{attribute 'GeneratedUsingTerminal: EK1122-0000-0018'}
{attribute addProperty BoxType "EK1122-0000-0018"}
{attribute addProperty Id "Term_17_EK1100Term_17_EK1100_E82441DC140"}
{attribute addProperty CRC "1353770864"}
{attribute addProperty Size "140"}
TYPE Term_16_EK1122_50B0E770 EXTENDS EK1122_1FC0878B :
STRUCT
	{attribute addProperty Name "Term_17_EK1100"}
	{attribute addProperty PreviousPort "Term 16 (EK1122) : D"}
	Term_17_EK1100 : Term_17_EK1100_E82441DC;
END_STRUCT
END_TYPE

(* stored: Version 1.2.0.0, ProductVersion 3.1.4024.9
   DUT Term_16_EK1122_50B0E770: Id {fa7c8029-8d97-0aa7-0914-3c2c5f2e586b} *)
